TYPE ST_ManualMode :
STRUCT
	bKeyPos : BOOL;
	bKeyNeg : BOOL;
	bKeyRapid : BOOL;
	nLogAxisNumber : UINT;
	nInc			: UINT;
	nManualTyp	: UINT;
	nSpeed : UINT;
	nHwResolution:	UDINT;    (* Handradauflösung in 0.1 um / Umdrehung *)
END_STRUCT
END_TYPE

(* stored: Version 1.1.0.1, ProductVersion 3.1.4022.12
   DUT ST_ManualMode: Id {90245e24-d94f-4fcb-8638-0dbe067658cd} *)
